(* Logix 5000 project; controller PBS_Perfusion vendor 1 type 14 code 217 rev 32.14; software revision 32.03 *)
// pbs perfusion / oxygenation skid

TASK CMs_100ms (periodic, rate 100 ms, priority 10, watchdog 500 ms) : CM_PBS
TASK PIDs_1000ms (periodic, rate 1000 ms, priority 10, watchdog 10000 ms) : PIDs

MODULES
   Local : vendor 1 type 14 code 217 (5069 0, rev 32.14)
      P101_Drive : ETHERNET-MODULE (Ethernet 192.168.1.30, rev 1.1, Output RPI 100 ms)   // stf stepper drive p101
      P103_Drive : ETHERNET-MODULE (Ethernet 192.168.1.32, rev 1.1, Output RPI 100 ms)   // stf stepper drive p103
      P104_Drive : ETHERNET-MODULE (Ethernet 192.168.1.33, rev 1.1, Output RPI 100 ms)   // stf stepper drive p104
      P102_Drive : ETHERNET-MODULE (Ethernet 192.168.1.31, rev 1.1, Output RPI 100 ms)   // stf stepper drive p102
      P105_Ethernet : 530_630_730 EtherNet/IP Pump (Ethernet 192.168.1.13, rev 2.5, StandardDataDriven RPI 20 ms)
           P105_Ethernet:I.FlowCal   // nl/rev
END_MODULES

TYPE AMP_Alarm_Word :   // Applied Motion Input Assembly - Alarm Word
STRUCT
   Position_Limit : BOOL;   // Position Limit
   CCW_Limit : BOOL;   // CCW Limit
   CW_Limit : BOOL;   // CW Limit
   Over_Temp : BOOL;   // Over Temp
   Excess_Regen_or_Internal_Voltage : BOOL;   // Excess Regen or Internal Voltage
   Over_Voltage : BOOL;   // Over Voltage
   Under_Voltage : BOOL;   // Under Voltage
   Over_Current : BOOL;   // Over Current
   Open_Motor_Windings : BOOL;   // Open Motor Windings
   Bad_Encoder : BOOL;   // Bad Encoder
   Comm_Error : BOOL;   // Comm Error
   Bad_Flash : BOOL;   // Bad Flash
   No_Move : BOOL;   // No Move
   NA_1 : BOOL;   // NA 1
   Blank_Q_Segment : BOOL;   // Blank Q Segment
   NA_2 : BOOL;   // NA 2
END_STRUCT
END_TYPE

TYPE AMP_Input_Assembly_v2 :   // Applied Motion Drive Input Assembly Version 2.0
STRUCT
   Status_Code : DINT;   // Status Code
   Alarm_Code : DINT;   // Alarm Code
   Voltage : DINT;   // Supply Voltage (x0.1V)
   Current : DINT;   // Actual Current (mA)
   Temp : DINT;   // Drive Temperature (0.1 deg C)
   Encoder_Position : DINT;   // Encoder Position (20,000 counts = 1 shaft turn)
   Absolute_Position : DINT;   // Absolute Position (20,000 counts = 1 shaft turn)
   Position_Error : DINT;   // Position Error (counts)
   Actual_Velocity : DINT;   // Actual Velocity (rev/sec * 240, 0 when no encoder)
   Extended_Inputs : DINT;   // Input Status (Extended)
   Main_Board_Inputs : DINT;   // Input Status (Main board)
   Word11 : DINT;   // Reserved
   Analog_Input_1 : DINT;   // Analog Input 1 (ADC counts, 0=min V, 16383 = max V)
   Analog_Input_2 : DINT;   // Analog Input 2 (ADC counts, 0=min V, 16383 = max V)
END_STRUCT
END_TYPE

TYPE AMP_Status_Word :   // Applied Motion Input Assembly Status Word
STRUCT
   Enabled : BOOL;   // Motor Enabled (Motor Disabled if this bit = 0)
   Sampling : BOOL;   // Sampling (for Quick Tuner)
   Drive_Fault : BOOL;   // Drive Fault (check Alarm Code)
   In_Position : BOOL;   // In Position (motor is in position)
   Moving : BOOL;   // Moving (motor is moving)
   Jogging : BOOL;   // Jogging (currently in jog mode)
   Stopping : BOOL;   // Stopping (in the process of stopping from a stop command)
   Waiting : BOOL;   // Waiting (for an input; executing a WI command)
   Saving : BOOL;   // Saving (parameter data is being saved)
   Alarm_Present : BOOL;   // Alarm present (check Alarm Code)
   Homing : BOOL;   // Homing (executing an SH command)
   Wait_Time : BOOL;   // Waiting (for time; executing a WD or WT command)
   Wizard_Running : BOOL;   // Wizard running (Timing Wizard is running)
   Checking_Encoder : BOOL;   // Checking encoder (Timing Wizard is running)
   Q_Program_Running : BOOL;   // Q Program is running
   Initializing : BOOL;   // Initializing (happens at power up) ; Servo Ready (for SV200 drives only)
END_STRUCT
END_TYPE

TYPE P_DescList :   // Code / Description List Entry
STRUCT
   Code : DINT;   // Code for which to look up Description
   Desc : STRING_40;   // Description for given Code
END_STRUCT
END_TYPE

TYPE PBSdata_UDT :
STRUCT
   agitation_pv : REAL;   // AgPV(RPM)
   agitation_sp : REAL;   // AgSP(RPM)
   agitation_man : REAL;   // AgPowerUser(%)
   agitation_mode : INT;   // AgModeUser
   agitation_error : INT;   // N/A: 0 means sensor is good and within range 40 means Low (corresponds to Agitation Low alarm) 50 means High (corresponds to Agitation High alarm) 90 means Low Low (corresponds to Agitation Low Low alarm) 100 means High High (corresponds to Agitation High High alarm) 200 means Fail (corresponds to Agitation Sensor Failure alarm)
   agitation_interlocked : INT;   // InterlockAgMotor
   agitation_output : REAL;   // AgPowerActualRequest(%)
   temperature_pv : REAL;   // TempPV(C)
   temperature_sp : REAL;   // TempSP(C)
   temperature_man : REAL;   // TempHeatDutyUser(%)
   temperature_mode : INT;   // TempModeUser
   temperature_error : INT;   // N/A: 0 means sensor is good and within range 40 means Low (corresponds to Temperature Low alarm) 50 means High (corresponds to Temperature High alarm) 90 means Low Low (corresponds to Temperature Low Low alarm) 100 means High High (corresponds to Temperature High High alarm) 200 means Fail (corresponds to Temp Sensor A Failure (range) alarm)
   temperature_interlocked : INT;   // InterlockHeater
   temperature_output : REAL;   // TempHeatDutyActual(%)
   do_pv : REAL;   // DOPV(%)
   do_sp : REAL;   // DOSP(%)
   do_manUp : REAL;   // DOO2FlowUser(%)
   do_manDown : REAL;   // DON2FlowUser(%)
   do_mode : INT;   // DOModeUser
   do_error : INT;   // N/A: 0 means sensor is good and within range 40 means Low (corresponds to DO Low alarm) 50 means High (corresponds to DO High alarm) 90 means Low Low (corresponds to DO Low Low alarm) 100 means High High (corresponds to DO High High alarm) 200 means Fail (corresponds to DO Sensor A Failure (range) alarm)
   do_interlocked : INT;   // InterlockGasFlow
   do_outputUp : REAL;   // DOO2FlowControllerRequestLimited(%)
   do_outputDown : REAL;   // DON2FlowActualRequest(%)
   ph_pv : REAL;   // pHPV
   ph_sp : REAL;   // pHSP
   ph_manUp : REAL;   // pHBaseDutyUser(%)
   ph_manDown : REAL;   // pHCO2User(%)
   ph_mode : INT;   // pHModeUser
   ph_error : INT;   // N/A: 0 means sensor is good and within range 40 means Low (corresponds to pH Low alarm) 50 means High (corresponds to pH High alarm) 90 means Low Low (corresponds to pH Low Low alarm) 100 means High High (corresponds to pH High High alarm) 200 means Fail (corresponds to either pH Sensor A Failure (range) alarm, or pH Sensor A Failure (rate) alarm)
   ph_interlocked : INT;   // InterlockGasFlow + InterlockPumps
   ph_outputUp : REAL;   // pHBaseDutyActual(%)
   ph_outputDown : REAL;   // pHCO2ActualRequest(%)
   pressure_pv : REAL;   // PressurePV(psi)
   pressure_error : INT;   // N/A: 0 means sensor is good and within range 40 means Low (corresponds to Pressure Low alarm) 50 means High (corresponds to Pressure High alarm) 90 means Low Low (corresponds to Pressure Low Low alarm) 100 means High High (corresponds to Pressure High High alarm) 200 means Fail (corresponds to Pressure Sensor Disconnected alarm)
   level_pv : REAL;   // LevelPV(L)
   level_error : INT;   // 0 means sensor is good and within range 40 means Low (corresponds to Level Low alarm) 50 means High (corresponds to Level High alarm) 90 means Low Low (corresponds to Level Low Low alarm) 100 means High High (corresponds to Level High High alarm) 200 is not applicable for Level
   condenser_pv : REAL;   // FilterOvenPV(C)
   condenser_sp : INT;   // FilterOvenSP(C)
   condenser_man : REAL;   // FilterOvenDutyUser(%)
   condenser_mode : INT;   // FilterOvenModeUser
   condenser_error : INT;   // N/A: 0 means sensor is good and within range 40 means Low (corresponds to Filter Oven Low alarm) 50 means High (corresponds to Filter Oven High alarm) 90 means Low Low (corresponds to Filter Oven Low Low alarm) 100 means High High (corresponds to Filter Oven High High alarm) 200 means Fail (no corresponding alarm)
   condenser_output : REAL;   // FilterOvenDutyActual(%)
   maingas_pv : REAL;   // MainGasFeedback(LPM)
   maingas_man : REAL;   // MainGasUser(LPM)
   maingas_mode : INT;   // MainGasModeUser
   maingas_error : INT;   // 0 means sensor is good and within range 40 means Low (corresponds to Main Gas Low alarm) 50 means High (corresponds to Main Gas High alarm) 90 means Low Low (corresponds to Main Gas Low Low alarm) 100 means High High (corresponds to Main Gas High High alarm) 200 is not applicable for Main Gas
   maingas_interlocked : INT;   // InterlockGasFlow
   MFCs_air : REAL;   // MFCAirFlowFeedback(LPM)
   MFCs_co2 : REAL;   // MFCCO2FlowFeedback(LPM)
   MFCs_n2 : REAL;   // MFCN2FlowFeedback(LPM)
   MFCs_o2 : REAL;   // MFCO2FlowFeedback(LPM)
   exchangeHeartbeat : BOOL;   // Heartbeat between the API exchange and PLC. If not flipping at specified rate, check console app is running
   jsonFailure : BOOL;   // If (1) API exchange can't reach webserver.
END_STRUCT
END_TYPE

TYPE STRING_12 :
STRUCT
   LEN : DINT;
   DATA : SINT[12];
END_STRUCT
END_TYPE

TYPE STRING_16 :
STRUCT
   LEN : DINT;
   DATA : SINT[16];
END_STRUCT
END_TYPE

TYPE STRING_20 :
STRUCT
   LEN : DINT;
   DATA : SINT[20];
END_STRUCT
END_TYPE

TYPE STRING_40 :
STRUCT
   LEN : DINT;
   DATA : SINT[40];
END_STRUCT
END_TYPE

TYPE STRING_8 :
STRUCT
   LEN : DINT;
   DATA : SINT[8];
END_STRUCT
END_TYPE

TYPE STRING_Area :
STRUCT
   LEN : DINT;
   DATA : SINT[8];
END_STRUCT
END_TYPE

TYPE STRING_Cond :
STRUCT
   LEN : DINT;
   DATA : SINT[20];
END_STRUCT
END_TYPE

TYPE STRING_NavTag :   // Navigation Tag
STRUCT
   LEN : DINT;
   DATA : SINT[20];
END_STRUCT
END_TYPE

ADD_ON_INSTRUCTION AMP_Alarm_Code   (* revision 1.0 *)
// Applied Motion - Alarm Code - AOI
// Help:
// The Alarm Code AOI uses the raw data stored in the Alarm Code word (Element 1 from Input Assembly 0x65) to set individual appropriately named boolean outputs.
VAR_INPUT
   Input : DINT; {required}   // Element 1 from Drive Input Assembly (0x65)
END_VAR
VAR_OUTPUT
   Position_Limit : BOOL; {access Read Only, visible}
   CCW_Limit : BOOL; {access Read Only, visible}
   CW_Limit : BOOL; {access Read Only, visible}
   Over_Temp : BOOL; {access Read Only, visible}
   Excess_Regen_or_Internal_Voltage : BOOL; {access Read Only, visible}
   Over_Voltage : BOOL; {access Read Only, visible}
   Under_Voltage : BOOL; {access Read Only, visible}
   Over_Current : BOOL; {access Read Only, visible}
   Open_Motor_Windings : BOOL; {access Read Only, visible}
   Bad_Encoder : BOOL; {access Read Only, visible}
   Comm_Error : BOOL; {access Read Only, visible}
   Bad_Flash : BOOL; {access Read Only, visible}
   No_Move : BOOL; {access Read Only, visible}
   NA_1 : BOOL; {access Read Only, visible}
   Blank_Q_Segment : BOOL; {access Read Only, visible}
   NA_2 : BOOL; {access Read Only, visible}
END_VAR

ROUTINE Logic   (* ladder *)
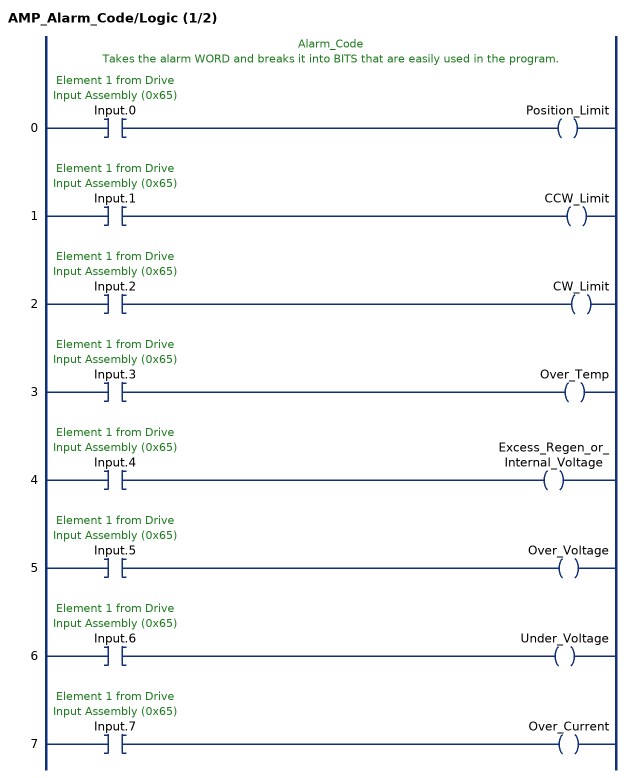
   // Alarm_Code
   // Takes the alarm WORD and breaks it into BITS that are easily used in the program.
   0: XIC(Input.0)OTE(Position_Limit);
   1: XIC(Input.1)OTE(CCW_Limit);
   2: XIC(Input.2)OTE(CW_Limit);
   3: XIC(Input.3)OTE(Over_Temp);
   4: XIC(Input.4)OTE(Excess_Regen_or_Internal_Voltage);
   5: XIC(Input.5)OTE(Over_Voltage);
   6: XIC(Input.6)OTE(Under_Voltage);
   7: XIC(Input.7)OTE(Over_Current);
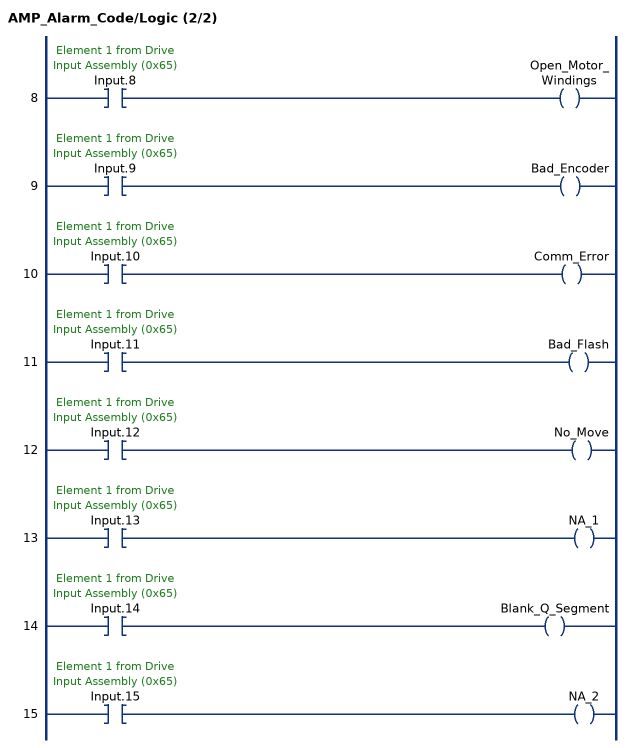
   8: XIC(Input.8)OTE(Open_Motor_Windings);
   9: XIC(Input.9)OTE(Bad_Encoder);
   10: XIC(Input.10)OTE(Comm_Error);
   11: XIC(Input.11)OTE(Bad_Flash);
   12: XIC(Input.12)OTE(No_Move);
   13: XIC(Input.13)OTE(NA_1);
   14: XIC(Input.14)OTE(Blank_Q_Segment);
   15: XIC(Input.15)OTE(NA_2);
END_ROUTINE
END_ADD_ON_INSTRUCTION

ADD_ON_INSTRUCTION AMP_Alarm_Reset   (* revision 1.0 *)
// Applied Motion - Alarm Reset - AOI
// Help:
// The Alarm Reset AOI is used to reset Drive Fault and clear Alarm Code (if possible). Figure 1 shows a preview of an instance of the AOI.
VAR_IN_OUT
   Input : DINT[14]; {required}   // Drive Input Assembly
   Output : DINT[16]; {required}   // Drive Output Assembly
        [0]   // Command Word
        [1]   // Jog Speed (0.25 rev/min)
        [2]   // Jog Acceleration (10 rev/s/s)
        [3]   // Jog Deceleration (10 rev/s/s)
        [4]   // Point-to-Point Velocity (0.25 rev/min)
        [5]   // Point-to-Point Acceleration (10 rev/s/s)
        [6]   // Point-to-Point Deceleration (10 rev/s/s)
        [7]   // Point-to-Point Distance (Motor steps)
        [9]   // (2x ASCII Letters in 16 lower word)
        [10]   // Data/Register 1
        [11]   // Data/Register 2
END_VAR
VAR_INPUT
   RPI : DINT := 100; {visible}   // Drive Connection Request Packet Interval (milliseconds)
   Reset : BOOL; {required}   // Reset the Drive (on rising edge)
END_VAR
VAR_OUTPUT
   Sent : BOOL; {access Read Only, visible}   // Reset has been sent to drive
   In_Progress : BOOL; {access Read Only, visible}   // Reset in progress
   Done : BOOL; {access Read Only, visible}   // Reset completed without errors - Drive is not faulted
   Error : BOOL; {access Read Only, visible}   // Reset failed - Not Used
   State : DINT := 10; {access None}   // Internal state of progress
END_VAR
VAR
   Loc_StatusCode : AMP_Status_Word;
   Loc_CommandOff_Timer : TIMER;   // Timer to make sure command value was 0 before sending a new command
   Loc_CommandOn_Timer : TIMER;   // Timer to make sure command value is set long enough to be sent to servo
   Loc_Input_Assembly : AMP_Input_Assembly_v2; {access None}
   Loc_Stop_ONS : BOOL; {access None}
END_VAR

ROUTINE Logic   (* ladder *)
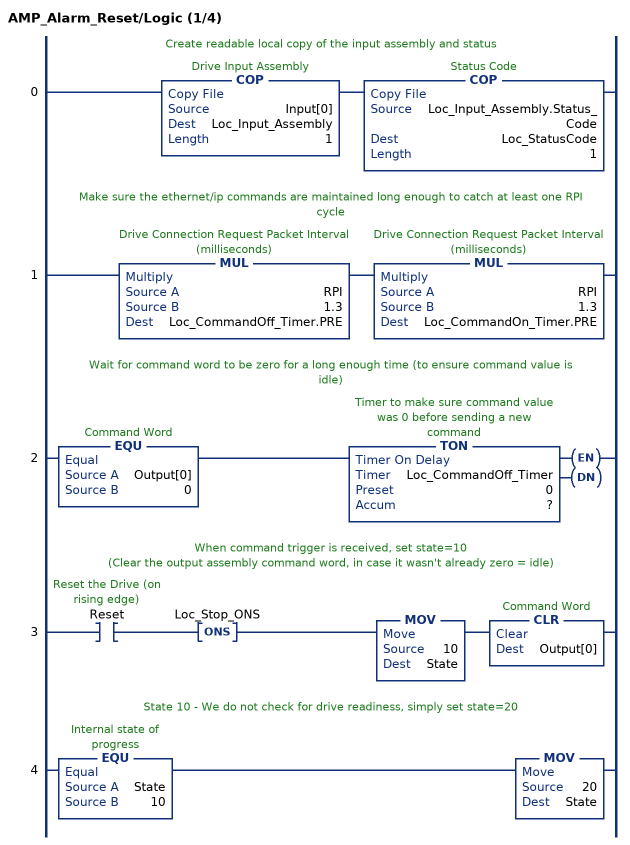
   // Create readable local copy of the input assembly and status
   0: COP(Input[0],Loc_Input_Assembly,1)COP(Loc_Input_Assembly.Status_Code,Loc_StatusCode,1);
   // Make sure the ethernet/ip commands are maintained long enough to catch at least one RPI cycle
   1: MUL(RPI,1.3,Loc_CommandOff_Timer.PRE)MUL(RPI,1.3,Loc_CommandOn_Timer.PRE);
   // Wait for command word to be zero for a long enough time (to ensure command value is idle)
   2: EQU(Output[0],0)TON(Loc_CommandOff_Timer,?,?);
   // When command trigger is received, set state=10
   // (Clear the output assembly command word, in case it wasn't already zero = idle)
   3: XIC(Reset)ONS(Loc_Stop_ONS)MOV(10,State)CLR(Output[0]);
   // State 10 - We do not check for drive readiness, simply set state=20
   4: EQU(State,10)MOV(20,State);
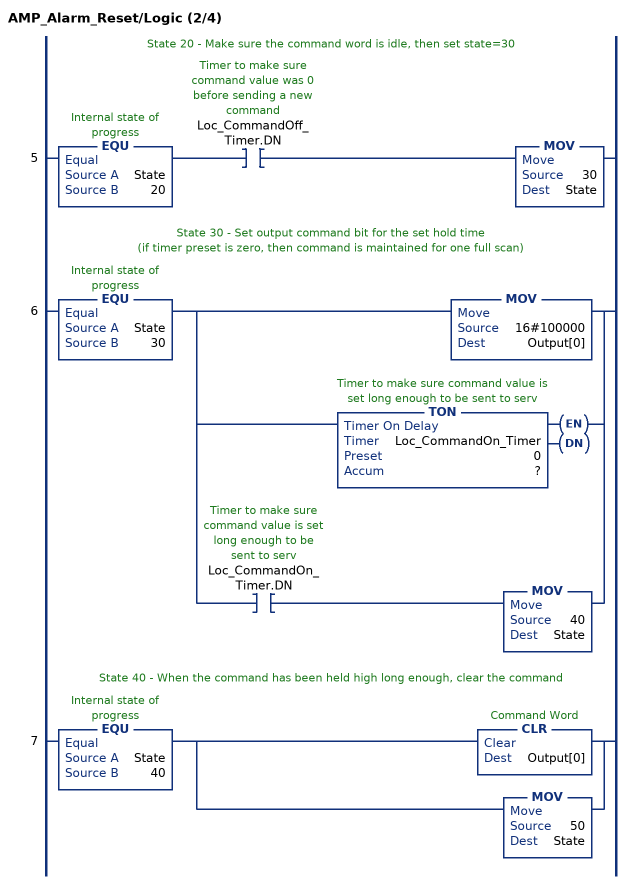
   // State 20 - Make sure the command word is idle, then set state=30
   5: EQU(State,20)XIC(Loc_CommandOff_Timer.DN)MOV(30,State);
   // State 30 - Set output command bit for the set hold time
   // (if timer preset is zero, then command is maintained for one full scan)
   6: EQU(State,30)[MOV(16#100000,Output[0]) ,TON(Loc_CommandOn_Timer,?,?) ,XIC(Loc_CommandOn_Timer.DN) MOV(40,State) ];
   // State 40 - When the command has been held high long enough, clear the command
   7: EQU(State,40)[CLR(Output[0]) ,MOV(50,State) ];
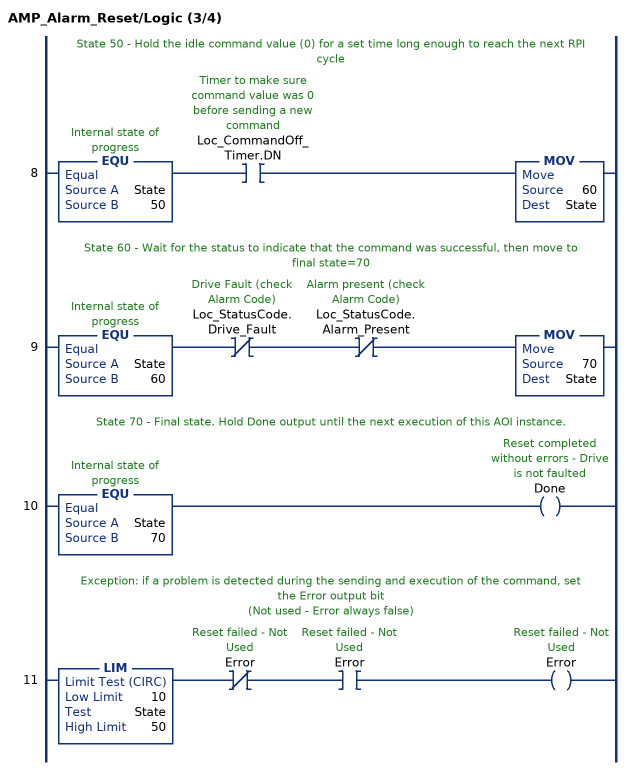
   // State 50 - Hold the idle command value (0) for a set time long enough to reach the next RPI cycle
   8: EQU(State,50)XIC(Loc_CommandOff_Timer.DN)MOV(60,State);
   // State 60 - Wait for the status to indicate that the command was successful, then move to final state=70
   9: EQU(State,60)XIO(Loc_StatusCode.Drive_Fault)XIO(Loc_StatusCode.Alarm_Present)MOV(70,State);
   // State 70 - Final state. Hold Done output until the next execution of this AOI instance.
   10: EQU(State,70)OTE(Done);
   // Exception: if a problem is detected during the sending and execution of the command, set the Error output bit
   // (Not used - Error always false)
   11: LIM(10,State,50)XIO(Error)XIC(Error)OTE(Error);
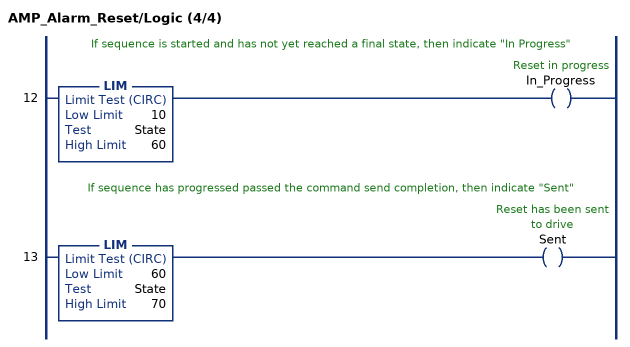
   // If sequence is started and has not yet reached a final state, then indicate "In Progress"
   12: LIM(10,State,60)OTE(In_Progress);
   // If sequence has progressed passed the command send completion, then indicate "Sent"
   13: LIM(60,State,70)OTE(Sent);
END_ROUTINE
END_ADD_ON_INSTRUCTION

ADD_ON_INSTRUCTION AMP_Configuration_Settings   (* revision 1.0 *)
// Applied Motion - Configuration Settings AOI
// Help:
// The Configuration Settings AOI accepts all the required parameters for: Position Fault (PF), Control Mode (CM), Secondary Control Mode (CN), Electronic Gearing (EG), Input Noise Filter (EI), Jerk Filter (KJ), and then scales and issues these to the drive, one at a time.
VAR_IN_OUT
   MSG_Write : SINT[8]; {required}   // Message Write data tag
        [0]   // Message Reserved = 0
        [1]   // Message Type (16#01 or 16#02)
        [2]   // Type 1: Register Type 2: Opcode
        [3]   // Type 1: Opcode Type 2: Operand
        [4]   // Type 1: Parameter 1 Type 2: data MSB
        [5]   // Type 1: Parameter 2 Type 2: data LSB
        [6]   // Type 1: Parameter 3 Type 2: not used
        [7]   // Type 1: Parameter 4 Type 2: not used
   SendMsg : MESSAGE; {required}   // Message tag
   MSG_Response : SINT[8]; {required}   // Message Response data tag
        [0]   // Command Word
        [1]   // Jog Speed (0.25 rev/min)
        [2]   // Jog Acceleration (10 rev/s/s)
        [3]   // Jog Deceleration (10 rev/s/s)
        [4]   // Point-to-Point Velocity (0.25 rev/min)
        [5]   // Point-to-Point Acceleration (10 rev/s/s)
        [6]   // Point-to-Point Deceleration (10 rev/s/s)
        [7]   // Point-to-Point Distance (Motor steps)
END_VAR
VAR_INPUT
   Configure : BOOL; {required}   // Start the Configuration
   PF : INT; {required}   // Position Fault (steps or counts)
   CM : INT; {required}   // Control Mode (integer code)
   CN : INT; {required}   // Secondary Control Mode (integer code)
   EG : INT; {required}   // Electronic Gearing (steps/rev or counts/rev)
   EI : INT; {required}   // Input Noise Filter Constant (0-255)
   KJ : INT; {required}   // Jerk Filter (Hz)
END_VAR
VAR_OUTPUT
   Sent : BOOL; {access Read Only, visible}   // All configuration settings have been sent to drive
   In_Progress : BOOL; {access Read Only, visible}   // The configuration is in progress
   Done : BOOL; {access Read Only, visible}   // Configuration completed without errors
   Error : BOOL; {access Read Only, visible}   // Configuration failed to complete - drive not ready or faulted
   State : DINT := 34; {access Read Only}   // Internal state of progress
END_VAR
VAR
   Loc_Start_ONS : BOOL; {access None}
   loc_Steps_per_Rev_div_by_2 : DINT;
END_VAR

ROUTINE Logic   (* ladder *)
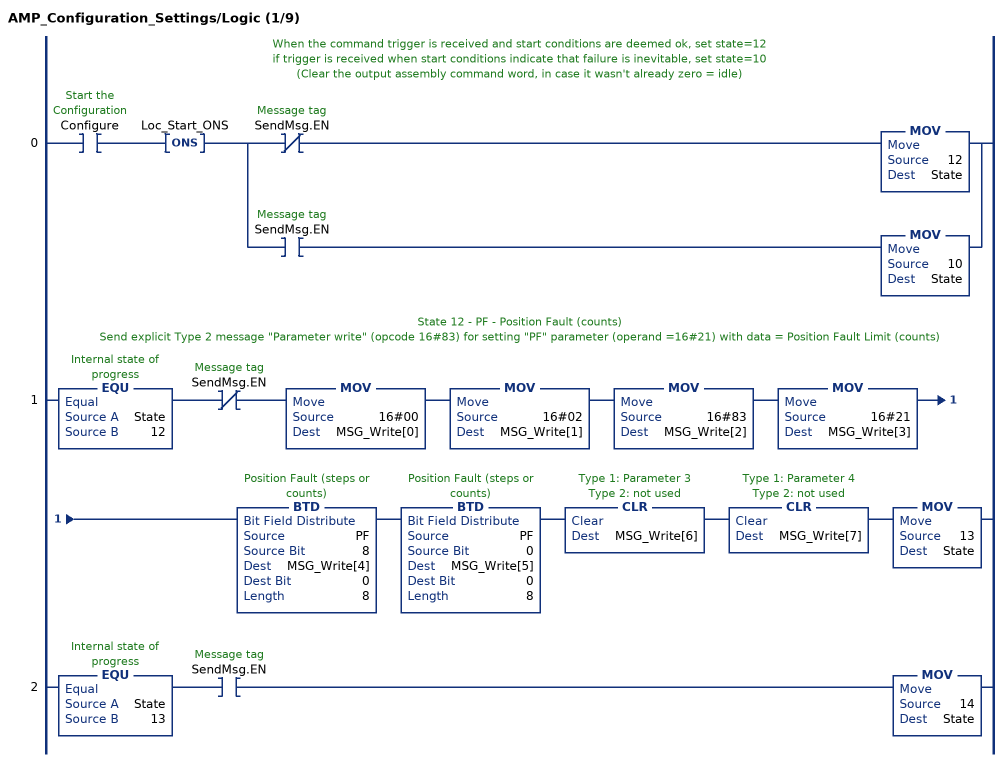
   // When the command trigger is received and start conditions are deemed ok, set state=12
   // if trigger is received when start conditions indicate that failure is inevitable, set state=10
   // (Clear the output assembly command word, in case it wasn't already zero = idle)
   0: XIC(Configure)ONS(Loc_Start_ONS)[XIO(SendMsg.EN) MOV(12,State) ,XIC(SendMsg.EN) MOV(10,State) ];
   // State 12 - PF - Position Fault (counts)
   // Send explicit Type 2 message "Parameter write" (opcode 16#83) for setting "PF" parameter (operand =16#21) with data = Position Fault Limit (counts)
   1: EQU(State,12)XIO(SendMsg.EN)MOV(16#00,MSG_Write[0])MOV(16#02,MSG_Write[1])MOV(16#83,MSG_Write[2])MOV(16#21,MSG_Write[3])BTD(PF,8,MSG_Write[4],0,8)BTD(PF,0,MSG_Write[5],0,8)CLR(MSG_Write[6])CLR(MSG_Write[7])MOV(13,State);
   2: EQU(State,13)XIC(SendMsg.EN)MOV(14,State);
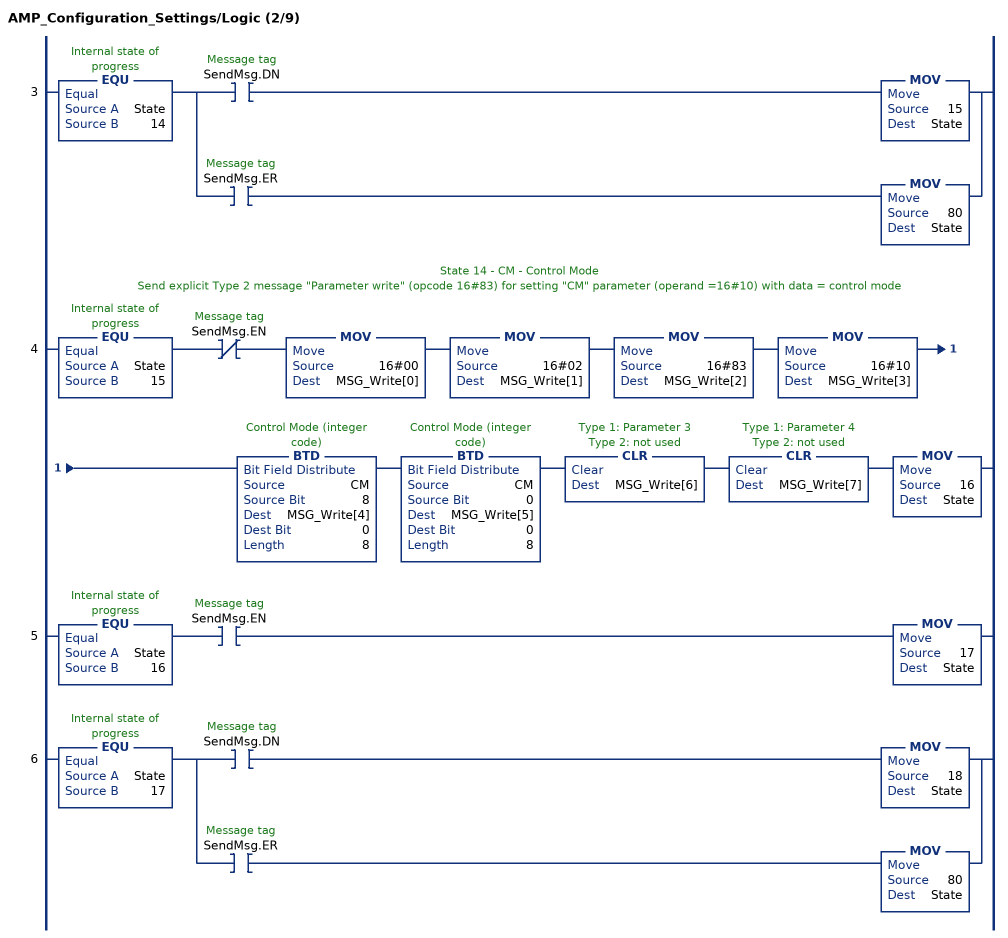
   3: EQU(State,14)[XIC(SendMsg.DN) MOV(15,State) ,XIC(SendMsg.ER) MOV(80,State) ];
   // State 14 - CM - Control Mode
   // Send explicit Type 2 message "Parameter write" (opcode 16#83) for setting "CM" parameter (operand =16#10) with data = control mode
   4: EQU(State,15)XIO(SendMsg.EN)MOV(16#00,MSG_Write[0])MOV(16#02,MSG_Write[1])MOV(16#83,MSG_Write[2])MOV(16#10,MSG_Write[3])BTD(CM,8,MSG_Write[4],0,8)BTD(CM,0,MSG_Write[5],0,8)CLR(MSG_Write[6])CLR(MSG_Write[7])MOV(16,State);
   5: EQU(State,16)XIC(SendMsg.EN)MOV(17,State);
   6: EQU(State,17)[XIC(SendMsg.DN) MOV(18,State) ,XIC(SendMsg.ER) MOV(80,State) ];
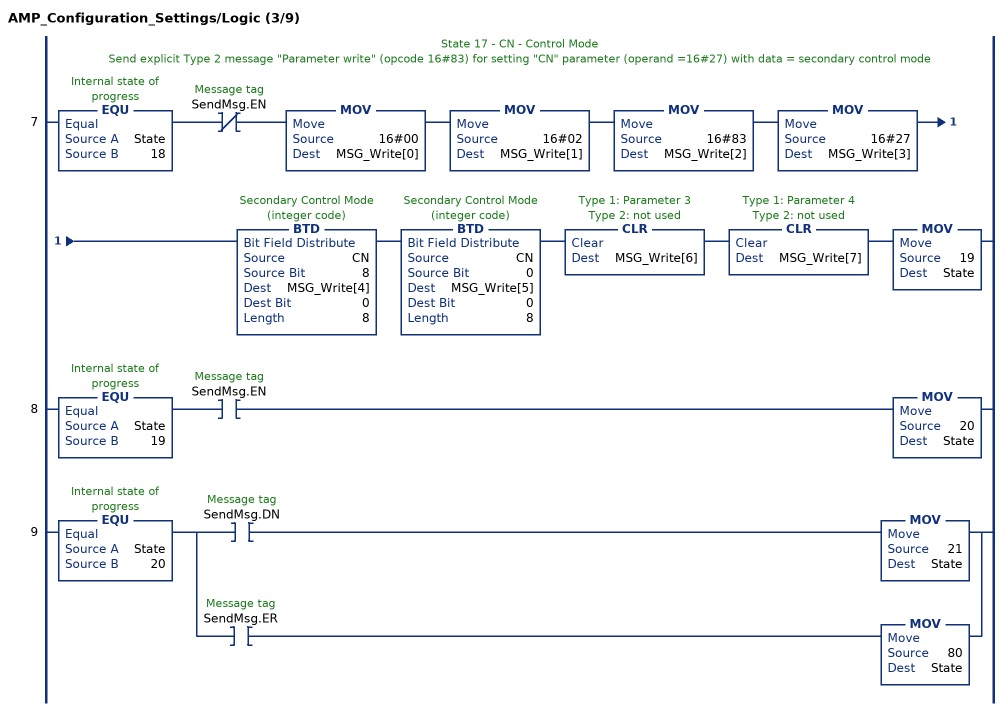
   // State 17 - CN - Control Mode
   // Send explicit Type 2 message "Parameter write" (opcode 16#83) for setting "CN" parameter (operand =16#27) with data = secondary control mode
   7: EQU(State,18)XIO(SendMsg.EN)MOV(16#00,MSG_Write[0])MOV(16#02,MSG_Write[1])MOV(16#83,MSG_Write[2])MOV(16#27,MSG_Write[3])BTD(CN,8,MSG_Write[4],0,8)BTD(CN,0,MSG_Write[5],0,8)CLR(MSG_Write[6])CLR(MSG_Write[7])MOV(19,State);
   8: EQU(State,19)XIC(SendMsg.EN)MOV(20,State);
   9: EQU(State,20)[XIC(SendMsg.DN) MOV(21,State) ,XIC(SendMsg.ER) MOV(80,State) ];
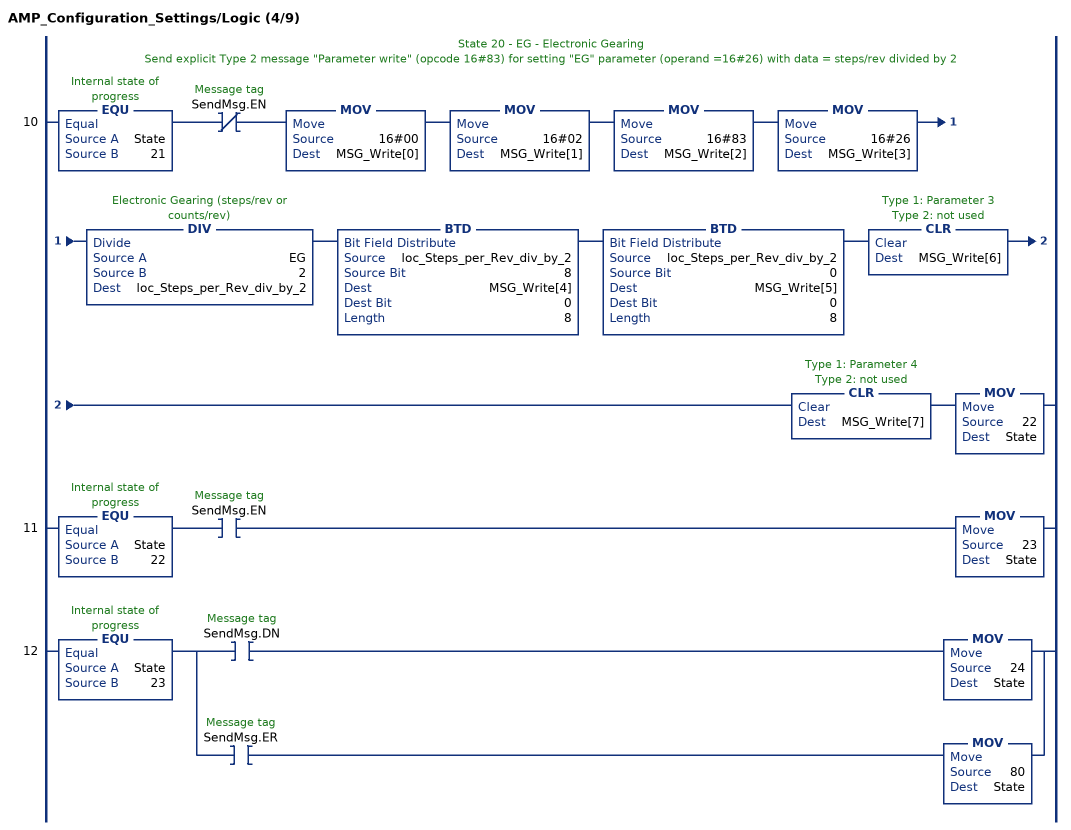
   // State 20 - EG - Electronic Gearing
   // Send explicit Type 2 message "Parameter write" (opcode 16#83) for setting "EG" parameter (operand =16#26) with data = steps/rev divided by 2
   10: EQU(State,21)XIO(SendMsg.EN)MOV(16#00,MSG_Write[0])MOV(16#02,MSG_Write[1])MOV(16#83,MSG_Write[2])MOV(16#26,MSG_Write[3])DIV(EG,2,loc_Steps_per_Rev_div_by_2)BTD(loc_Steps_per_Rev_div_by_2,8,MSG_Write[4],0,8)BTD(loc_Steps_per_Rev_div_by_2,0,MSG_Write[5],0,8)CLR(MSG_Write[6])CLR(MSG_Write[7])MOV(22,State);
   11: EQU(State,22)XIC(SendMsg.EN)MOV(23,State);
   12: EQU(State,23)[XIC(SendMsg.DN) MOV(24,State) ,XIC(SendMsg.ER) MOV(80,State) ];
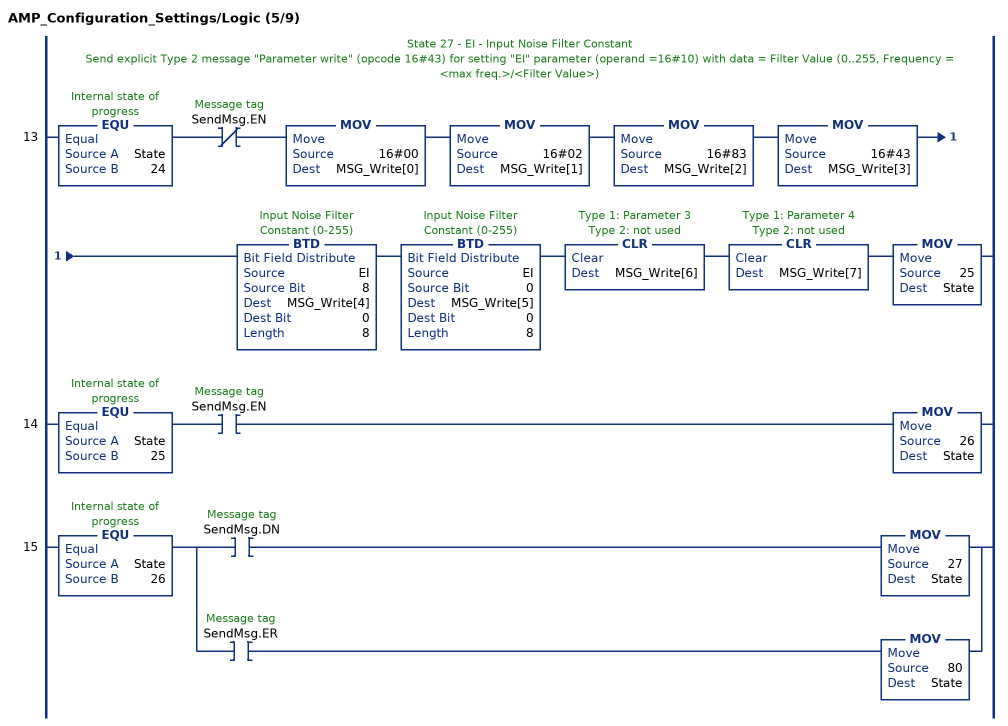
   // State 27 - EI - Input Noise Filter Constant
   // Send explicit Type 2 message "Parameter write" (opcode 16#43) for setting "EI" parameter (operand =16#10) with data = Filter Value (0..255, Frequency = <max freq.>/<Filter Value>)
   13: EQU(State,24)XIO(SendMsg.EN)MOV(16#00,MSG_Write[0])MOV(16#02,MSG_Write[1])MOV(16#83,MSG_Write[2])MOV(16#43,MSG_Write[3])BTD(EI,8,MSG_Write[4],0,8)BTD(EI,0,MSG_Write[5],0,8)CLR(MSG_Write[6])CLR(MSG_Write[7])MOV(25,State);
   14: EQU(State,25)XIC(SendMsg.EN)MOV(26,State);
   15: EQU(State,26)[XIC(SendMsg.DN) MOV(27,State) ,XIC(SendMsg.ER) MOV(80,State) ];
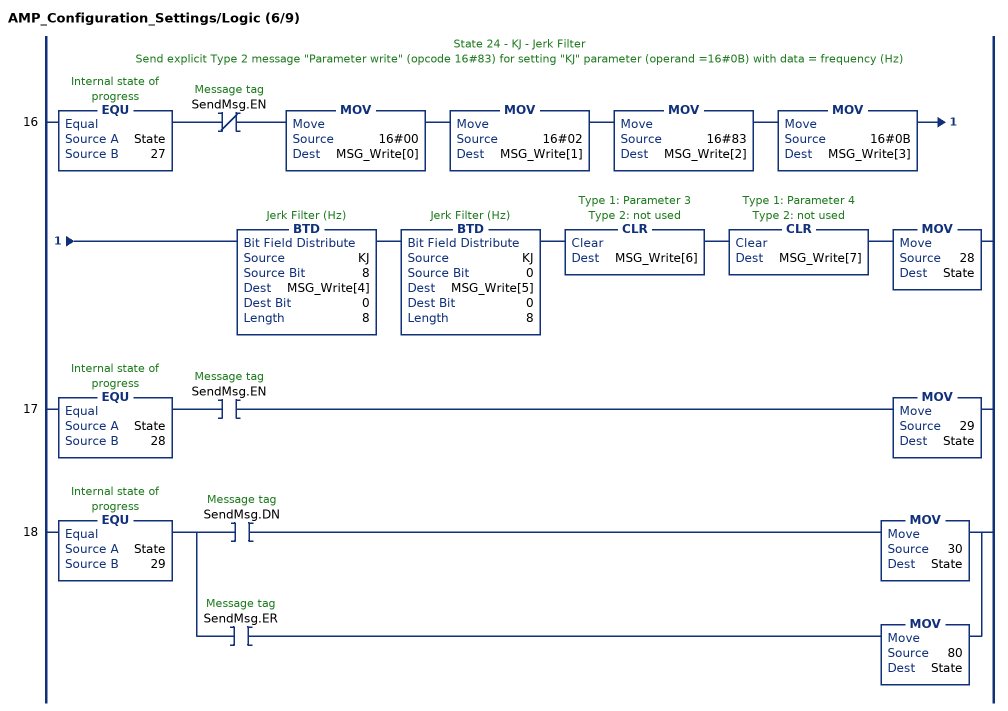
   // State 24 - KJ - Jerk Filter
   // Send explicit Type 2 message "Parameter write" (opcode 16#83) for setting "KJ" parameter (operand =16#0B) with data = frequency (Hz)
   16: EQU(State,27)XIO(SendMsg.EN)MOV(16#00,MSG_Write[0])MOV(16#02,MSG_Write[1])MOV(16#83,MSG_Write[2])MOV(16#0B,MSG_Write[3])BTD(KJ,8,MSG_Write[4],0,8)BTD(KJ,0,MSG_Write[5],0,8)CLR(MSG_Write[6])CLR(MSG_Write[7])MOV(28,State);
   17: EQU(State,28)XIC(SendMsg.EN)MOV(29,State);
   18: EQU(State,29)[XIC(SendMsg.DN) MOV(30,State) ,XIC(SendMsg.ER) MOV(80,State) ];
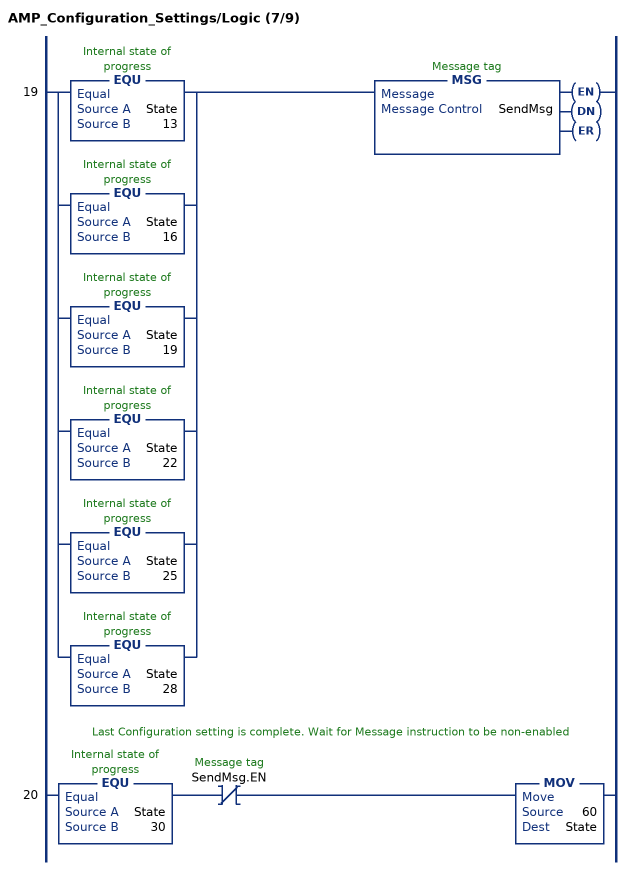
   19: [EQU(State,13) ,EQU(State,16) ,EQU(State,19) ,EQU(State,22) ,EQU(State,25) ,EQU(State,28) ]MSG(SendMsg);
   // Last Configuration setting is complete. Wait for Message instruction to be non-enabled
   20: EQU(State,30)XIO(SendMsg.EN)MOV(60,State);
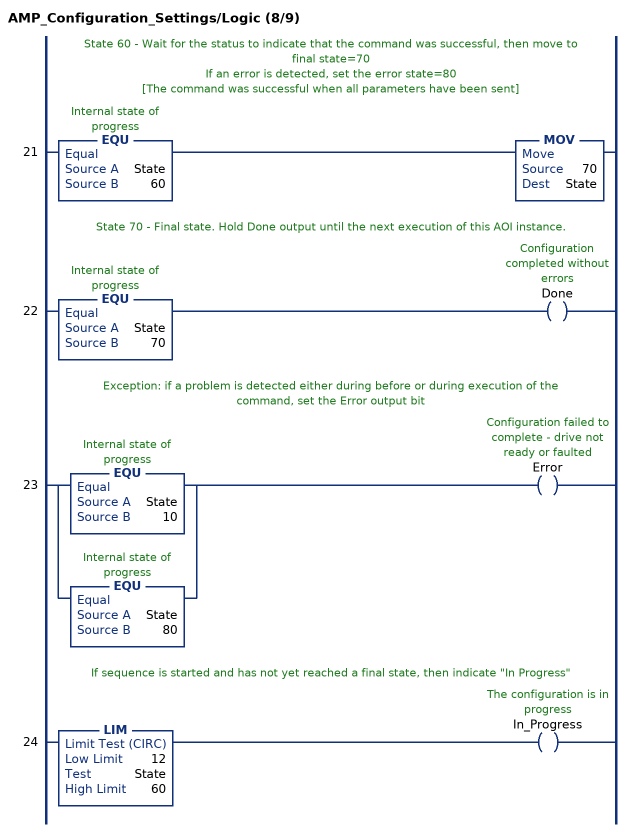
   // State 60 - Wait for the status to indicate that the command was successful, then move to final state=70
   // If an error is detected, set the error state=80
   // [The command was successful when all parameters have been sent]
   21: EQU(State,60)MOV(70,State);
   // State 70 - Final state. Hold Done output until the next execution of this AOI instance.
   22: EQU(State,70)OTE(Done);
   // Exception: if a problem is detected either during before or during execution of the command, set the Error output bit
   23: [EQU(State,10) ,EQU(State,80) ]OTE(Error);
   // If sequence is started and has not yet reached a final state, then indicate "In Progress"
   24: LIM(12,State,60)OTE(In_Progress);
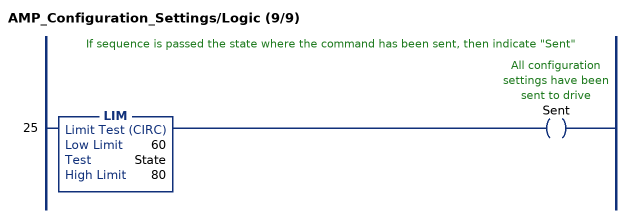
   // If sequence is passed the state where the command has been sent, then indicate "Sent"
   25: LIM(60,State,80)OTE(Sent);
END_ROUTINE
END_ADD_ON_INSTRUCTION

ADD_ON_INSTRUCTION AMP_Crash_Stop   (* revision 1.0 *)
// Applied Motion - Stop/Kill using Maximum Deceleration - AOI
// Help:
// The Crash Stop AOI is used to stop and kill the drive using the maximum deceleration as set by the AM command.
VAR_IN_OUT
   Input : DINT[14]; {required}   // Drive Input Assembly
   Output : DINT[16]; {required}   // Drive Output Assembly
        [0]   // Command Word
        [1]   // Jog Speed (0.25 rev/min)
        [2]   // Jog Acceleration (10 rev/s/s)
        [3]   // Jog Deceleration (10 rev/s/s)
        [4]   // Point-to-Point Velocity (0.25 rev/min)
        [5]   // Point-to-Point Acceleration (10 rev/s/s)
        [6]   // Point-to-Point Deceleration (10 rev/s/s)
        [7]   // Point-to-Point Distance (Motor steps)
        [9]   // (2x ASCII Letters in 16 lower word)
        [10]   // Data/Register 1
        [11]   // Data/Register 2
END_VAR
VAR_INPUT
   RPI : DINT := 100; {visible}   // Drive Connection Request Packet Interval (milliseconds)
   Stop : BOOL; {required}   // Stop the drive axis
END_VAR
VAR_OUTPUT
   Sent : BOOL; {access Read Only, visible}   // Stop has been sent to drive
   In_Progress : BOOL; {access Read Only, visible}   // Stop in progress
   Done : BOOL; {access Read Only, visible}   // Stop completed without errors - Servo is not moving
   Error : BOOL; {access Read Only, visible}   // Stop failed - drive not ready or faulted
   State : DINT := 10; {access None}   // Internal state of progress
END_VAR
VAR
   Loc_StatusCode : AMP_Status_Word;
   Loc_CommandOff_Timer : TIMER;   // Timer to make sure command value was 0 before sending a new command
   Loc_CommandOn_Timer : TIMER;   // Timer to make sure command value is set long enough to be sent to servo
   Loc_Input_Assembly : AMP_Input_Assembly_v2; {access None}
   Loc_Stop_ONS : BOOL; {access None}
END_VAR

ROUTINE Logic   (* ladder *)
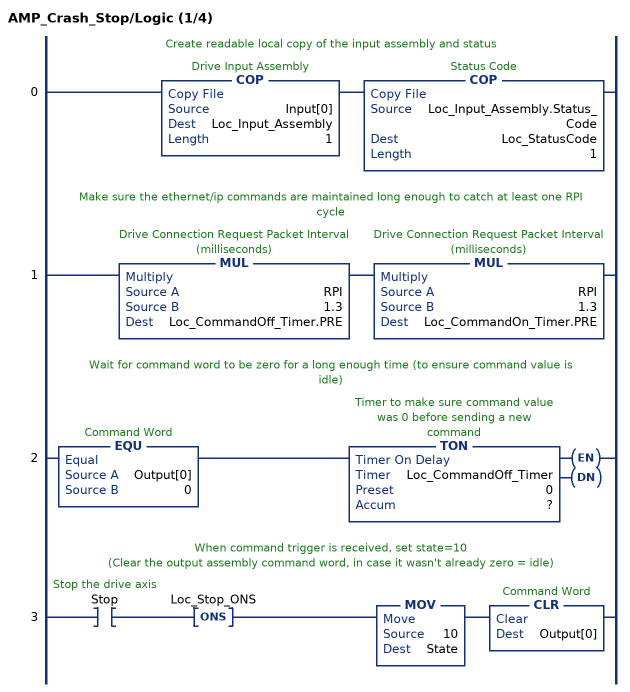
   // Create readable local copy of the input assembly and status
   0: COP(Input[0],Loc_Input_Assembly,1)COP(Loc_Input_Assembly.Status_Code,Loc_StatusCode,1);
   // Make sure the ethernet/ip commands are maintained long enough to catch at least one RPI cycle
   1: MUL(RPI,1.3,Loc_CommandOff_Timer.PRE)MUL(RPI,1.3,Loc_CommandOn_Timer.PRE);
   // Wait for command word to be zero for a long enough time (to ensure command value is idle)
   2: EQU(Output[0],0)TON(Loc_CommandOff_Timer,?,?);
   // When command trigger is received, set state=10
   // (Clear the output assembly command word, in case it wasn't already zero = idle)
   3: XIC(Stop)ONS(Loc_Stop_ONS)MOV(10,State)CLR(Output[0]);
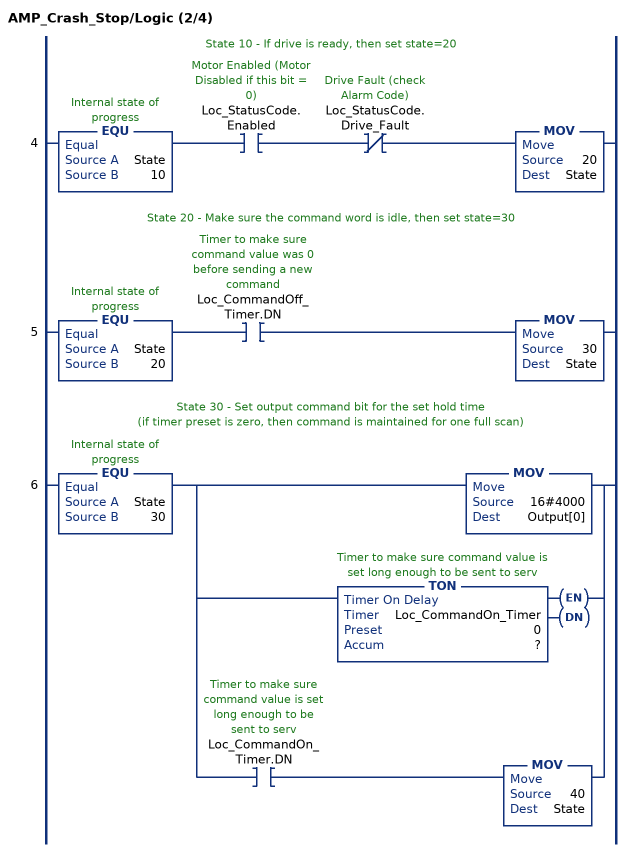
   // State 10 - If drive is ready, then set state=20
   4: EQU(State,10)XIC(Loc_StatusCode.Enabled)XIO(Loc_StatusCode.Drive_Fault)MOV(20,State);
   // State 20 - Make sure the command word is idle, then set state=30
   5: EQU(State,20)XIC(Loc_CommandOff_Timer.DN)MOV(30,State);
   // State 30 - Set output command bit for the set hold time
   // (if timer preset is zero, then command is maintained for one full scan)
   6: EQU(State,30)[MOV(16#4000,Output[0]) ,TON(Loc_CommandOn_Timer,?,?) ,XIC(Loc_CommandOn_Timer.DN) MOV(40,State) ];
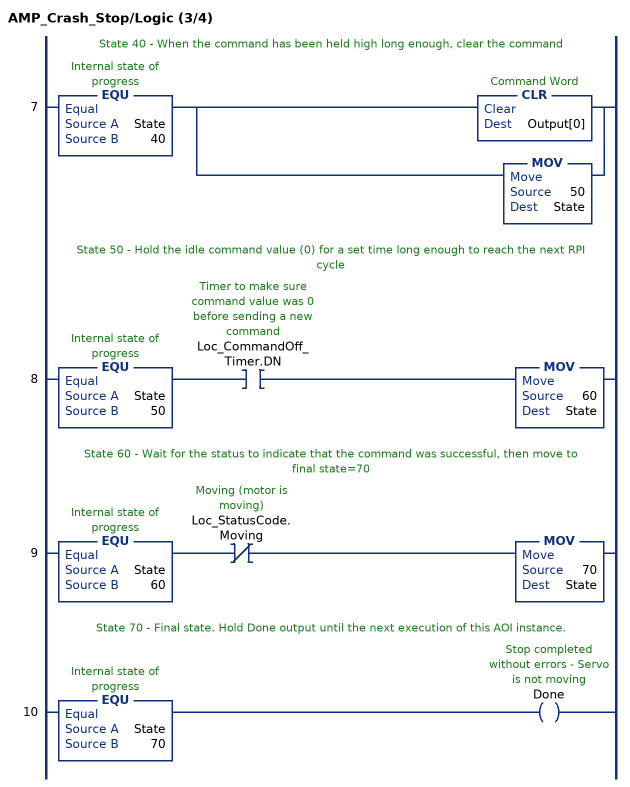
   // State 40 - When the command has been held high long enough, clear the command
   7: EQU(State,40)[CLR(Output[0]) ,MOV(50,State) ];
   // State 50 - Hold the idle command value (0) for a set time long enough to reach the next RPI cycle
   8: EQU(State,50)XIC(Loc_CommandOff_Timer.DN)MOV(60,State);
   // State 60 - Wait for the status to indicate that the command was successful, then move to final state=70
   9: EQU(State,60)XIO(Loc_StatusCode.Moving)MOV(70,State);
   // State 70 - Final state. Hold Done output until the next execution of this AOI instance.
   10: EQU(State,70)OTE(Done);
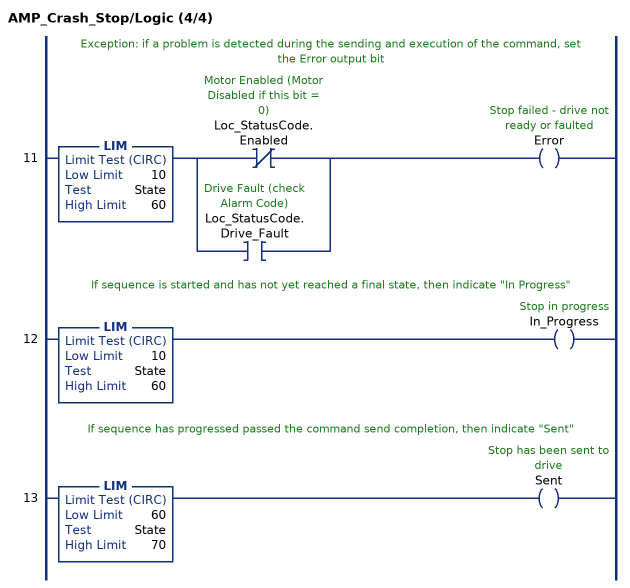
   // Exception: if a problem is detected during the sending and execution of the command, set the Error output bit
   11: LIM(10,State,60)[XIO(Loc_StatusCode.Enabled) ,XIC(Loc_StatusCode.Drive_Fault) ]OTE(Error);
   // If sequence is started and has not yet reached a final state, then indicate "In Progress"
   12: LIM(10,State,60)OTE(In_Progress);
   // If sequence has progressed passed the command send completion, then indicate "Sent"
   13: LIM(60,State,70)OTE(Sent);
END_ROUTINE
END_ADD_ON_INSTRUCTION
